(****************************************************************
NAME:			FB_SetPhaseLowerAxisPosition
DATA:			2022.10.18
VERSION:		1.0.0
DESCRIPTION:	FB_SetPhaseLowerAxisPosition
HISTORY:
				2022.10.18		NEW

***************************************************************)
FUNCTION_BLOCK FB_SetPhaseLowerMotorAxisPosition
VAR_INPUT
	ValueSet:LREAL:=0;
	Execute:BOOL;
END_VAR
VAR_OUTPUT
	FbID:DINT:=1001;
	State:DINT;
	Busy:BOOL;
	Done:BOOL;
	Error:BOOL;
	ErrorID:DINT;
END_VAR
VAR
	PhaseLowerMotor_MC_SetPosition: MC_SetPosition;
	fb_ton: TON;
	FB_PlcEmergencyStop: FB_PlcEmergencyStop;
END_VAR

IF Execute THEN
Busy:=TRUE;
Done:=FALSE;
fb_ton(PT:=t#0.1s);
CASE State OF
	0:
		IF PhaseLowerMotor_MC_SetPosition.Error THEN		(*FB Error*)
			ErrorID:=1;
			State:=99;
		ELSE
			State:=1;
		END_IF
	1:	(*Execute*)
		PhaseLowerMotor_MC_SetPosition.Position:=ValueSet;
		PhaseLowerMotor_MC_SetPosition.Execute:=TRUE;
		A_SetPhaseLowerPositionMC();
		fb_ton.IN:=TRUE;
		State:=2;
	2:	(*Wait*)
		A_SetPhaseLowerPositionMC();
		IF NOT PhaseLowerMotor_MC_SetPosition.Done THEN		
			IF NOT fb_ton.Q THEN
				State:=2;
			ELSE
				ErrorID:=4;
				State:=99;
			END_IF
		ELSIF  PhaseLowerMotor_MC_SetPosition.Done THEN	
			State:=88;
		ELSE
			ErrorID:=5;
			State:=99;
		END_IF
	88:
		Execute:=FALSE;
		State:=0;
		Busy:=FALSE;
		Done:=TRUE;
		Error:=FALSE;
		ErrorID:=0;
		PhaseLowerMotor_MC_SetPosition.Execute:=FALSE;
		fb_ton.IN:=FALSE;
	99:
		Execute:=FALSE;
		State:=99;
		Busy:=FALSE;
		Done:=FALSE;
		Error:=TRUE;
		PhaseLowerMotor_MC_SetPosition.Execute:=FALSE;
		fb_ton.IN:=FALSE;
	-100:
		FB_PlcEmergencyStop();
		Execute:=FALSE;
		State:=-100;
		Busy:=FALSE;
		Done:=FALSE;
		Error:=TRUE;
		PhaseLowerMotor_MC_SetPosition.Execute:=FALSE;
		fb_ton.IN:=FALSE;
END_CASE
END_IF

ACTION A_SetPhaseLowerPositionMC:
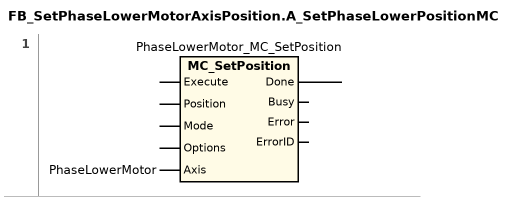
// NETWORK 1
PhaseLowerMotor_MC_SetPosition(Axis := PhaseLowerMotor); // MC_SetPosition
END_ACTION

END_FUNCTION_BLOCK

(* stored: Version 1.1.0.1, ProductVersion 3.1.4024.6
   POU FB_SetPhaseLowerMotorAxisPosition: Id {8e7eee3a-8fda-4d2b-a3aa-d33a0f1377b2}, SpecialFunc None
   Action A_SetPhaseLowerPositionMC: Id {33f63e16-473c-4566-a3eb-a0d60b324d81} *)
